// TIA Portal V21 export
FUNCTION "GestStazione_AbilitaDestinazione" : Void   // FC412, LAD
{ S7_Optimized_Access := 'TRUE' }
// stored: SetENOAutomatically false
   VAR_INPUT
      K_StazioneSorgente : Int;
      K_StazioneDestinazione : Int;
   END_VAR
BEGIN

REGION Network 1
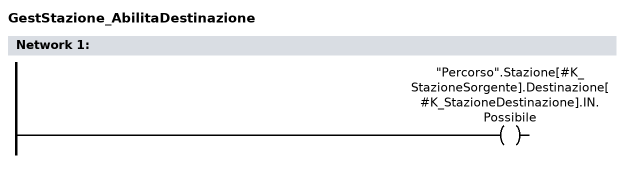
   RUNG wire#powerrail
      Coil( "Percorso".Stazione[#K_StazioneSorgente].Destinazione[#K_StazioneDestinazione].IN.Possibile )
   END_RUNG
   // the same network as SCL:
   "Percorso".Stazione[#K_StazioneSorgente].Destinazione[#K_StazioneDestinazione].IN.Possibile := TRUE;
END_REGION
END_FUNCTION
